// TwinCAT 3 PLC project Untitled1
// ProgramVersion: 3.1.4024.0
// libraries:
//   Tc2_Standard, * (Beckhoff Automation GmbH)
//   Tc2_System, * (Beckhoff Automation GmbH)
//   Tc3_Module, * (Beckhoff Automation GmbH)
// project tree:
//   GVLs/ GVL.TcGVL
//   / PlcTask.TcTTO, Task1_1.TcTTO, Task2_1.TcTTO
//   POUs/ task1.TcPOU, Task2.TcPOU
// real-time tasks:
//   TASK PlcTask: cycle T#10ms, priority 20, ADS port 350
//   TASK Task1: cycle T#10ms, priority 21, ADS port 351
//   TASK Task2: cycle T#10ms, priority 22, ADS port 352

CONFIGURATION Untitled1
    RESOURCE PLC ON TwinCAT3
        TASK PlcTask(INTERVAL := T#10ms, PRIORITY := 20);
        TASK Task1_1(INTERVAL := T#10ms, PRIORITY := 21);
        TASK Task2_1(INTERVAL := T#10ms, PRIORITY := 22);
        PROGRAM task1 WITH Task1_1 : task1;
        PROGRAM Task2 WITH Task2_1 : Task2;
    END_RESOURCE
END_CONFIGURATION

// ---- GVLs/GVL.TcGVL
VAR_GLOBAL
    bInDeventer : BOOL := FALSE;      // Reiziger is in Deventer
    bKoffieGereed : BOOL := FALSE;    // Koffie is gehaald door koffietaak
    sStatusTekst : STRING := '';      // Status voor visualisatie
END_VAR

// ---- POUs/task1.TcPOU
PROGRAM task1
VAR
	PRG_Reis: INT;
	bReisGestart: BOOL;
END_VAR

// Start de reis
IF NOT bReisGestart THEN
    bReisGestart := TRUE;
    sStatusTekst := 'Ik ben onderweg naar Deventer...';
END_IF

// Aankomst in Deventer
IF bReisGestart AND NOT bInDeventer THEN
    bInDeventer := TRUE;
    sStatusTekst := 'Ik ben in Deventer. Ik wacht op koffie...';
END_IF

// Wachten op koffie van Task 2
IF bInDeventer AND bKoffieGereed THEN
    sStatusTekst := 'Koffie ontvangen! Ik reis door naar school.';
END_IF

END_PROGRAM

// ---- POUs/Task2.TcPOU
PROGRAM Task2
VAR
	PRG_Koffie: INT;
	bKoffieStart: BOOL;
END_VAR

// Start koffie-proces alleen als we in Deventer zijn
IF bInDeventer AND NOT bKoffieStart THEN
    bKoffieStart := TRUE;
    sStatusTekst := 'Koffie halen is gestart...';
END_IF

// Koffie ophalen (simulatie)
IF bKoffieStart THEN
    bKoffieGereed := TRUE;
    sStatusTekst := 'Koffie is gehaald!';
END_IF

END_PROGRAM
